// TIA Portal V17 export
// export: Created 2025-03-05T08:02:54.8462086Z, ExportSetting WithDefaults, DisplayName Totally Integrated Automation Portal, DisplayVersion V17 Update 8, DisplayName TIA Portal Openness, DisplayVersion V17 Update 8, DisplayName TIA Portal Version Control Interface, DisplayVersion V17, DisplayName SINAMICS Startdrive Advanced, DisplayVersion V17 SP2, DisplayName SINAMICS Startdrive G110M, G120, G120C, G120D, G120P, G115D, DisplayVersion V17 SP2, DisplayName SINAMICS Startdrive G130, G150, S120, S150, SINAMICS MV, S210, DisplayVersion V17 SP2, DisplayName STEP 7 Professional, DisplayVersion V17 Update 8, DisplayName SINUMERIK ONE STEP 7 Toolbox, DisplayVersion V17 Update 12, DisplayName SINUMERIK 840D sl STEP 7 Toolbox, DisplayVersion V17 Update 12, DisplayName STEP 7 Safety, DisplayVersion V17 Update 6, DisplayName WinCC Advanced, DisplayVersion V17 Update 8
DATA_BLOCK "DB7238_VARIABLES_PLC_CONNECTION"   // DB7238
{ S7_Optimized_Access := 'TRUE'; DB_Accessible_From_OPC_UA := 'FALSE' }
VERSION : 0.1
// stored: AutoNumber false, DBAccessibleFromOPCUA false, DBAccessibleFromWebserver true, IsOnlyStoredInLoadMemory false, IsRetainMemResEnabled false, IsWriteProtectedInAS false, MemoryReserve 100
   VAR RETAIN
      FEEDER_1_U_01_LINE_1 { S7_SetPoint := 'True'} : "UDT_Feeder Line";
      FEEDER_1_U_01_LINE_2 { S7_SetPoint := 'True'} : "UDT_Feeder Line";
      FEEDER_1_U_02_LINE_1 { S7_SetPoint := 'True'} : "UDT_Feeder Line";
      FEEDER_1_U_02_LINE_2 { S7_SetPoint := 'True'} : "UDT_Feeder Line";
      FEEDER_2_U_02_LINE_1 { S7_SetPoint := 'True'} : "UDT_Feeder Line";
      FEEDER_2_U_02_LINE_2 { S7_SetPoint := 'True'} : "UDT_Feeder Line";
      HOPPER_U_01_LINE_1 { S7_SetPoint := 'True'} : "UDT_Hopper Line";
      HOPPER_U_01_LINE_2 { S7_SetPoint := 'True'} : "UDT_Hopper Line";
      HOPPER_U_02_LINE_1 { S7_SetPoint := 'True'} : "UDT_Hopper Line";
      HOPPER_U_02_LINE_2 { S7_SetPoint := 'True'} : "UDT_Hopper Line";
   END_VAR
   VAR
      HOPPER_U_02_LINE_3 { S7_SetPoint := 'True'} : "UDT_Hopper Line";
      GENERAL : Struct
         PLC_TO_HMI : Struct
            FEEDERS_MODE_STATE : Int := 1;   // FEEDERS MODE STATE (1= AUTO. 3= MANUAL)
            HOPPERS_MODE_STATE : Int := 1;   // HOPPERS MODE STATE (1= AUTO. 3= MANUAL)
         END_STRUCT;
         HMI_TO_PLC : Struct
            FEEDERS_AUTO_MODE : Bool := FALSE;   // FEEDERS AUTO MODE HMI BUTTON
            FEEDERS_MANUAL_MODE : Bool := FALSE;   // FEEDERS MANUAL MODE HMI BUTTON
            HOPPERS_AUTO_MODE : Bool := FALSE;   // HOPPERS AUTO MODE HMI BUTTON
            HOPPERS_MANUAL_MODE : Bool := FALSE;   // HOPPERS MANUAL MODE HMI BUTTON
         END_STRUCT;
      END_STRUCT;
   END_VAR
   VAR RETAIN
      SELECTED_UNIT { S7_SetPoint := 'True'} : Int := 0;
      FEEDER_1_U01_SELECTED_GAS : Int := 1;   // SELECTED GAS. 1 = ARGON. 2 = NITROGEN. 3 = HELIUM. 4 = ARGON30
   END_VAR
   VAR
      FEEDER_1_U01_CHANGE_GAS_COND : Bool;   // CHANGE GAS CONDITIONS
   END_VAR
   VAR RETAIN
      FEEDER_1_U02_SELECTED_GAS : Int := 1;   // SELECTED GAS. 1 = ARGON. 2 = NITROGEN. 3 = HELIUM. 4 = ARGON30
   END_VAR
   VAR
      FEEDER_1_U02_CHANGE_GAS_COND : Bool;   // CHANGE GAS CONDITIONS
   END_VAR
   VAR RETAIN
      FEEDER_2_U02_SELECTED_GAS : Int := 1;   // SELECTED GAS. 1 = ARGON. 2 = NITROGEN. 3 = HELIUM. 4 = ARGON30
   END_VAR
   VAR
      FEEDER_2_U02_CHANGE_GAS_COND : Bool;   // CHANGE GAS CONDITIONS
      CURRENT_PROTECTION_LEVEL : Byte := 16#01;   // CURRENT ACCESS LEVEL
      EKS_USER : String := 'ETX4   $07';   // EKS OPERATOR ID
      HMI_USER : String := 'Engineering';
      HMI_PASSWORD : WString := WSTRING#'Engineering';
      EKS_OPERATOR_IDENTIFICATION : Byte := 16#01;   // EKS OPERATOR IDENTIFICATION
   END_VAR
BEGIN
   FEEDER_1_U_01_LINE_1.GAS_FLOW_RATE_ACTUAL := 0.0;
   FEEDER_1_U_01_LINE_1.GAS_FLOW_RATE_AUTO := 11.0;
   FEEDER_1_U_01_LINE_1.GAS_FLOW_RATE_MANUAL := 10.0;
   FEEDER_1_U_01_LINE_1.DISC_SPEED_ACTUAL := 0.0;
   FEEDER_1_U_01_LINE_1.DISC_SPEED_AUTO := 44.0;
   FEEDER_1_U_01_LINE_1.DISC_SPEED_MANUAL := 44.0;
   FEEDER_1_U_01_LINE_1.STIRRER_SPEED_ACTUAL := 0.0;
   FEEDER_1_U_01_LINE_1.STIRRER_SPEED_AUTO := 30.0;
   FEEDER_1_U_01_LINE_1.STIRRER_SPEED_MANUAL := 30.0;
   FEEDER_1_U_01_LINE_1.HOPPER_TEMP_ACTUAL := -1.0;
   FEEDER_1_U_01_LINE_1.HOPPER_TEMP_AUTO := 0.0;
   FEEDER_1_U_01_LINE_1.HOPPER_TEMP_MANUAL := 0.0;
   FEEDER_1_U_01_LINE_1.HEATER_ON_MANUAL_REQUEST := FALSE;
   FEEDER_1_U_01_LINE_1.HEATER_OFF_MANUAL_REQUEST := FALSE;
   FEEDER_1_U_01_LINE_1.HOPPER_ON_MANUAL_REQUEST := FALSE;
   FEEDER_1_U_01_LINE_1.HOPPER_OFF_MANUAL_REQUEST := FALSE;
   FEEDER_1_U_01_LINE_1.HOPPER_STATUS := 16#00;
   FEEDER_1_U_01_LINE_1.START_SEQUENCE_GAS_STEPS := 5;
   FEEDER_1_U_01_LINE_1.START_SEQUENCE_DISK_STEPS := 5;
   FEEDER_1_U_01_LINE_1.STOP_SEQUENCE_GAS_STEPS := 10;
   FEEDER_1_U_01_LINE_1.STOP_SEQUENCE_DISK_STEPS := 10;
   FEEDER_1_U_01_LINE_1.STOP_SEQUENCE_PAUSE_STEP := 5;
   FEEDER_1_U_01_LINE_1.DISC_SPEED_WARNING_UPPER_LIMIT := 1.0;
   FEEDER_1_U_01_LINE_1.DISC_SPEED_ALARM_UPPER_LIMIT := 2.0;
   FEEDER_1_U_01_LINE_1.DISC_SPEED_WARNING_LOWER_LIMIT := 1.0;
   FEEDER_1_U_01_LINE_1.DISC_SPEED_ALARM_LOWER_LIMIT := 2.0;
   FEEDER_1_U_01_LINE_1.GAS_FLOW_RATE_WARNING_UPPER_LIMIT := 1.0;
   FEEDER_1_U_01_LINE_1.GAS_FLOW_RATE_ALARM_UPPER_LIMIT := 4.0;
   FEEDER_1_U_01_LINE_1.GAS_FLOW_RATE_WARNING_LOWER_LIMIT := 1.0;
   FEEDER_1_U_01_LINE_1.GAS_FLOW_RATE_ALARM_LOWER_LIMIT := 4.0;
   FEEDER_1_U_01_LINE_1.STIRRER_SPEED_WARNING_UPPER_LIMIT := 1.0;
   FEEDER_1_U_01_LINE_1.STIRRER_SPEED_ALARM_UPPER_LIMIT := 5.0;
   FEEDER_1_U_01_LINE_1.STIRRER_SPEED_WARNING_LOWER_LIMIT := 1.0;
   FEEDER_1_U_01_LINE_1.STIRRER_SPEED_ALARM_LOWER_LIMIT := 10.0;
   FEEDER_1_U_01_LINE_1.HOPPER_TEMP_ALARM_UPPER_LIMIT := 3.0;
   FEEDER_1_U_01_LINE_1.PRESSURE_VALUE_CURRENT_SENSOR := 0.0;
   FEEDER_1_U_01_LINE_2.GAS_FLOW_RATE_ACTUAL := 0.0;
   FEEDER_1_U_01_LINE_2.GAS_FLOW_RATE_AUTO := 11.0;
   FEEDER_1_U_01_LINE_2.GAS_FLOW_RATE_MANUAL := 10.0;
   FEEDER_1_U_01_LINE_2.DISC_SPEED_ACTUAL := 0.0;
   FEEDER_1_U_01_LINE_2.DISC_SPEED_AUTO := 44.0;
   FEEDER_1_U_01_LINE_2.DISC_SPEED_MANUAL := 44.0;
   FEEDER_1_U_01_LINE_2.STIRRER_SPEED_ACTUAL := 0.0;
   FEEDER_1_U_01_LINE_2.STIRRER_SPEED_AUTO := 30.0;
   FEEDER_1_U_01_LINE_2.STIRRER_SPEED_MANUAL := 30.0;
   FEEDER_1_U_01_LINE_2.HOPPER_TEMP_ACTUAL := -1.0;
   FEEDER_1_U_01_LINE_2.HOPPER_TEMP_AUTO := 0.0;
   FEEDER_1_U_01_LINE_2.HOPPER_TEMP_MANUAL := 0.0;
   FEEDER_1_U_01_LINE_2.HEATER_ON_MANUAL_REQUEST := FALSE;
   FEEDER_1_U_01_LINE_2.HEATER_OFF_MANUAL_REQUEST := FALSE;
   FEEDER_1_U_01_LINE_2.HOPPER_ON_MANUAL_REQUEST := FALSE;
   FEEDER_1_U_01_LINE_2.HOPPER_OFF_MANUAL_REQUEST := FALSE;
   FEEDER_1_U_01_LINE_2.HOPPER_STATUS := 16#00;
   FEEDER_1_U_01_LINE_2.START_SEQUENCE_GAS_STEPS := 5;
   FEEDER_1_U_01_LINE_2.START_SEQUENCE_DISK_STEPS := 5;
   FEEDER_1_U_01_LINE_2.STOP_SEQUENCE_GAS_STEPS := 10;
   FEEDER_1_U_01_LINE_2.STOP_SEQUENCE_DISK_STEPS := 10;
   FEEDER_1_U_01_LINE_2.STOP_SEQUENCE_PAUSE_STEP := 5;
   FEEDER_1_U_01_LINE_2.DISC_SPEED_WARNING_UPPER_LIMIT := 1.0;
   FEEDER_1_U_01_LINE_2.DISC_SPEED_ALARM_UPPER_LIMIT := 2.0;
   FEEDER_1_U_01_LINE_2.DISC_SPEED_WARNING_LOWER_LIMIT := 1.0;
   FEEDER_1_U_01_LINE_2.DISC_SPEED_ALARM_LOWER_LIMIT := 2.0;
   FEEDER_1_U_01_LINE_2.GAS_FLOW_RATE_WARNING_UPPER_LIMIT := 1.0;
   FEEDER_1_U_01_LINE_2.GAS_FLOW_RATE_ALARM_UPPER_LIMIT := 4.0;
   FEEDER_1_U_01_LINE_2.GAS_FLOW_RATE_WARNING_LOWER_LIMIT := 1.0;
   FEEDER_1_U_01_LINE_2.GAS_FLOW_RATE_ALARM_LOWER_LIMIT := 4.0;
   FEEDER_1_U_01_LINE_2.STIRRER_SPEED_WARNING_UPPER_LIMIT := 1.0;
   FEEDER_1_U_01_LINE_2.STIRRER_SPEED_ALARM_UPPER_LIMIT := 5.0;
   FEEDER_1_U_01_LINE_2.STIRRER_SPEED_WARNING_LOWER_LIMIT := 1.0;
   FEEDER_1_U_01_LINE_2.STIRRER_SPEED_ALARM_LOWER_LIMIT := 10.0;
   FEEDER_1_U_01_LINE_2.HOPPER_TEMP_ALARM_UPPER_LIMIT := 3.0;
   FEEDER_1_U_01_LINE_2.PRESSURE_VALUE_CURRENT_SENSOR := 0.0;
   FEEDER_1_U_02_LINE_1.GAS_FLOW_RATE_ACTUAL := 13.99967;
   FEEDER_1_U_02_LINE_1.GAS_FLOW_RATE_AUTO := 14.0;
   FEEDER_1_U_02_LINE_1.GAS_FLOW_RATE_MANUAL := 14.0;
   FEEDER_1_U_02_LINE_1.DISC_SPEED_ACTUAL := 78.12334;
   FEEDER_1_U_02_LINE_1.DISC_SPEED_AUTO := 78.0;
   FEEDER_1_U_02_LINE_1.DISC_SPEED_MANUAL := 77.0;
   FEEDER_1_U_02_LINE_1.STIRRER_SPEED_ACTUAL := 30.15667;
   FEEDER_1_U_02_LINE_1.STIRRER_SPEED_AUTO := 30.0;
   FEEDER_1_U_02_LINE_1.STIRRER_SPEED_MANUAL := 30.0;
   FEEDER_1_U_02_LINE_1.HOPPER_TEMP_ACTUAL := 17.4;
   FEEDER_1_U_02_LINE_1.HOPPER_TEMP_AUTO := 0.0;
   FEEDER_1_U_02_LINE_1.HOPPER_TEMP_MANUAL := 0.0;
   FEEDER_1_U_02_LINE_1.HEATER_ON_MANUAL_REQUEST := FALSE;
   FEEDER_1_U_02_LINE_1.HEATER_OFF_MANUAL_REQUEST := FALSE;
   FEEDER_1_U_02_LINE_1.HOPPER_ON_MANUAL_REQUEST := FALSE;
   FEEDER_1_U_02_LINE_1.HOPPER_OFF_MANUAL_REQUEST := FALSE;
   FEEDER_1_U_02_LINE_1.HOPPER_STATUS := 16#01;
   FEEDER_1_U_02_LINE_1.START_SEQUENCE_GAS_STEPS := 5;
   FEEDER_1_U_02_LINE_1.START_SEQUENCE_DISK_STEPS := 5;
   FEEDER_1_U_02_LINE_1.STOP_SEQUENCE_GAS_STEPS := 10;
   FEEDER_1_U_02_LINE_1.STOP_SEQUENCE_DISK_STEPS := 10;
   FEEDER_1_U_02_LINE_1.STOP_SEQUENCE_PAUSE_STEP := 5;
   FEEDER_1_U_02_LINE_1.DISC_SPEED_WARNING_UPPER_LIMIT := 10.0;
   FEEDER_1_U_02_LINE_1.DISC_SPEED_ALARM_UPPER_LIMIT := 2.0;
   FEEDER_1_U_02_LINE_1.DISC_SPEED_WARNING_LOWER_LIMIT := 15.0;
   FEEDER_1_U_02_LINE_1.DISC_SPEED_ALARM_LOWER_LIMIT := 2.0;
   FEEDER_1_U_02_LINE_1.GAS_FLOW_RATE_WARNING_UPPER_LIMIT := 3.0;
   FEEDER_1_U_02_LINE_1.GAS_FLOW_RATE_ALARM_UPPER_LIMIT := 4.0;
   FEEDER_1_U_02_LINE_1.GAS_FLOW_RATE_WARNING_LOWER_LIMIT := 15.0;
   FEEDER_1_U_02_LINE_1.GAS_FLOW_RATE_ALARM_LOWER_LIMIT := 4.0;
   FEEDER_1_U_02_LINE_1.STIRRER_SPEED_WARNING_UPPER_LIMIT := 10.0;
   FEEDER_1_U_02_LINE_1.STIRRER_SPEED_ALARM_UPPER_LIMIT := 5.0;
   FEEDER_1_U_02_LINE_1.STIRRER_SPEED_WARNING_LOWER_LIMIT := 99.0;
   FEEDER_1_U_02_LINE_1.STIRRER_SPEED_ALARM_LOWER_LIMIT := 10.0;
   FEEDER_1_U_02_LINE_1.HOPPER_TEMP_ALARM_UPPER_LIMIT := 0.0;
   FEEDER_1_U_02_LINE_1.PRESSURE_VALUE_CURRENT_SENSOR := 0.0;
   FEEDER_1_U_02_LINE_2.GAS_FLOW_RATE_ACTUAL := 13.99837;
   FEEDER_1_U_02_LINE_2.GAS_FLOW_RATE_AUTO := 14.0;
   FEEDER_1_U_02_LINE_2.GAS_FLOW_RATE_MANUAL := 14.0;
   FEEDER_1_U_02_LINE_2.DISC_SPEED_ACTUAL := 77.98333;
   FEEDER_1_U_02_LINE_2.DISC_SPEED_AUTO := 78.0;
   FEEDER_1_U_02_LINE_2.DISC_SPEED_MANUAL := 77.0;
   FEEDER_1_U_02_LINE_2.STIRRER_SPEED_ACTUAL := 29.89333;
   FEEDER_1_U_02_LINE_2.STIRRER_SPEED_AUTO := 30.0;
   FEEDER_1_U_02_LINE_2.STIRRER_SPEED_MANUAL := 30.0;
   FEEDER_1_U_02_LINE_2.HOPPER_TEMP_ACTUAL := 17.6;
   FEEDER_1_U_02_LINE_2.HOPPER_TEMP_AUTO := 0.0;
   FEEDER_1_U_02_LINE_2.HOPPER_TEMP_MANUAL := 0.0;
   FEEDER_1_U_02_LINE_2.HEATER_ON_MANUAL_REQUEST := FALSE;
   FEEDER_1_U_02_LINE_2.HEATER_OFF_MANUAL_REQUEST := FALSE;
   FEEDER_1_U_02_LINE_2.HOPPER_ON_MANUAL_REQUEST := FALSE;
   FEEDER_1_U_02_LINE_2.HOPPER_OFF_MANUAL_REQUEST := FALSE;
   FEEDER_1_U_02_LINE_2.HOPPER_STATUS := 16#01;
   FEEDER_1_U_02_LINE_2.START_SEQUENCE_GAS_STEPS := 5;
   FEEDER_1_U_02_LINE_2.START_SEQUENCE_DISK_STEPS := 5;
   FEEDER_1_U_02_LINE_2.STOP_SEQUENCE_GAS_STEPS := 10;
   FEEDER_1_U_02_LINE_2.STOP_SEQUENCE_DISK_STEPS := 10;
   FEEDER_1_U_02_LINE_2.STOP_SEQUENCE_PAUSE_STEP := 5;
   FEEDER_1_U_02_LINE_2.DISC_SPEED_WARNING_UPPER_LIMIT := 10.0;
   FEEDER_1_U_02_LINE_2.DISC_SPEED_ALARM_UPPER_LIMIT := 2.0;
   FEEDER_1_U_02_LINE_2.DISC_SPEED_WARNING_LOWER_LIMIT := 15.0;
   FEEDER_1_U_02_LINE_2.DISC_SPEED_ALARM_LOWER_LIMIT := 2.0;
   FEEDER_1_U_02_LINE_2.GAS_FLOW_RATE_WARNING_UPPER_LIMIT := 3.0;
   FEEDER_1_U_02_LINE_2.GAS_FLOW_RATE_ALARM_UPPER_LIMIT := 4.0;
   FEEDER_1_U_02_LINE_2.GAS_FLOW_RATE_WARNING_LOWER_LIMIT := 15.0;
   FEEDER_1_U_02_LINE_2.GAS_FLOW_RATE_ALARM_LOWER_LIMIT := 4.0;
   FEEDER_1_U_02_LINE_2.STIRRER_SPEED_WARNING_UPPER_LIMIT := 10.0;
   FEEDER_1_U_02_LINE_2.STIRRER_SPEED_ALARM_UPPER_LIMIT := 5.0;
   FEEDER_1_U_02_LINE_2.STIRRER_SPEED_WARNING_LOWER_LIMIT := 99.0;
   FEEDER_1_U_02_LINE_2.STIRRER_SPEED_ALARM_LOWER_LIMIT := 10.0;
   FEEDER_1_U_02_LINE_2.HOPPER_TEMP_ALARM_UPPER_LIMIT := 3.0;
   FEEDER_1_U_02_LINE_2.PRESSURE_VALUE_CURRENT_SENSOR := 0.0;
   FEEDER_2_U_02_LINE_1.GAS_FLOW_RATE_ACTUAL := 0.0;
   FEEDER_2_U_02_LINE_1.GAS_FLOW_RATE_AUTO := 0.0;
   FEEDER_2_U_02_LINE_1.GAS_FLOW_RATE_MANUAL := 0.0;
   FEEDER_2_U_02_LINE_1.DISC_SPEED_ACTUAL := 0.0;
   FEEDER_2_U_02_LINE_1.DISC_SPEED_AUTO := 0.0;
   FEEDER_2_U_02_LINE_1.DISC_SPEED_MANUAL := 0.0;
   FEEDER_2_U_02_LINE_1.STIRRER_SPEED_ACTUAL := 0.0;
   FEEDER_2_U_02_LINE_1.STIRRER_SPEED_AUTO := 0.0;
   FEEDER_2_U_02_LINE_1.STIRRER_SPEED_MANUAL := 0.0;
   FEEDER_2_U_02_LINE_1.HOPPER_TEMP_ACTUAL := 0.0;
   FEEDER_2_U_02_LINE_1.HOPPER_TEMP_AUTO := 0.0;
   FEEDER_2_U_02_LINE_1.HOPPER_TEMP_MANUAL := 0.0;
   FEEDER_2_U_02_LINE_1.HEATER_ON_MANUAL_REQUEST := FALSE;
   FEEDER_2_U_02_LINE_1.HEATER_OFF_MANUAL_REQUEST := FALSE;
   FEEDER_2_U_02_LINE_1.HOPPER_ON_MANUAL_REQUEST := FALSE;
   FEEDER_2_U_02_LINE_1.HOPPER_OFF_MANUAL_REQUEST := FALSE;
   FEEDER_2_U_02_LINE_1.HOPPER_STATUS := 16#00;
   FEEDER_2_U_02_LINE_1.START_SEQUENCE_GAS_STEPS := 0;
   FEEDER_2_U_02_LINE_1.START_SEQUENCE_DISK_STEPS := 0;
   FEEDER_2_U_02_LINE_1.STOP_SEQUENCE_GAS_STEPS := 0;
   FEEDER_2_U_02_LINE_1.STOP_SEQUENCE_DISK_STEPS := 0;
   FEEDER_2_U_02_LINE_1.STOP_SEQUENCE_PAUSE_STEP := 0;
   FEEDER_2_U_02_LINE_1.DISC_SPEED_WARNING_UPPER_LIMIT := 0.0;
   FEEDER_2_U_02_LINE_1.DISC_SPEED_ALARM_UPPER_LIMIT := 0.0;
   FEEDER_2_U_02_LINE_1.DISC_SPEED_WARNING_LOWER_LIMIT := 0.0;
   FEEDER_2_U_02_LINE_1.DISC_SPEED_ALARM_LOWER_LIMIT := 0.0;
   FEEDER_2_U_02_LINE_1.GAS_FLOW_RATE_WARNING_UPPER_LIMIT := 0.0;
   FEEDER_2_U_02_LINE_1.GAS_FLOW_RATE_ALARM_UPPER_LIMIT := 0.0;
   FEEDER_2_U_02_LINE_1.GAS_FLOW_RATE_WARNING_LOWER_LIMIT := 0.0;
   FEEDER_2_U_02_LINE_1.GAS_FLOW_RATE_ALARM_LOWER_LIMIT := 0.0;
   FEEDER_2_U_02_LINE_1.STIRRER_SPEED_WARNING_UPPER_LIMIT := 0.0;
   FEEDER_2_U_02_LINE_1.STIRRER_SPEED_ALARM_UPPER_LIMIT := 0.0;
   FEEDER_2_U_02_LINE_1.STIRRER_SPEED_WARNING_LOWER_LIMIT := 0.0;
   FEEDER_2_U_02_LINE_1.STIRRER_SPEED_ALARM_LOWER_LIMIT := 0.0;
   FEEDER_2_U_02_LINE_1.HOPPER_TEMP_ALARM_UPPER_LIMIT := 0.0;
   FEEDER_2_U_02_LINE_1.PRESSURE_VALUE_CURRENT_SENSOR := 0.0;
   FEEDER_2_U_02_LINE_2.GAS_FLOW_RATE_ACTUAL := 14.00755;
   FEEDER_2_U_02_LINE_2.GAS_FLOW_RATE_AUTO := 14.0;
   FEEDER_2_U_02_LINE_2.GAS_FLOW_RATE_MANUAL := 14.0;
   FEEDER_2_U_02_LINE_2.DISC_SPEED_ACTUAL := 44.02667;
   FEEDER_2_U_02_LINE_2.DISC_SPEED_AUTO := 44.0;
   FEEDER_2_U_02_LINE_2.DISC_SPEED_MANUAL := 77.0;
   FEEDER_2_U_02_LINE_2.STIRRER_SPEED_ACTUAL := 29.94667;
   FEEDER_2_U_02_LINE_2.STIRRER_SPEED_AUTO := 30.0;
   FEEDER_2_U_02_LINE_2.STIRRER_SPEED_MANUAL := 30.0;
   FEEDER_2_U_02_LINE_2.HOPPER_TEMP_ACTUAL := 17.4;
   FEEDER_2_U_02_LINE_2.HOPPER_TEMP_AUTO := 0.0;
   FEEDER_2_U_02_LINE_2.HOPPER_TEMP_MANUAL := 0.0;
   FEEDER_2_U_02_LINE_2.HEATER_ON_MANUAL_REQUEST := FALSE;
   FEEDER_2_U_02_LINE_2.HEATER_OFF_MANUAL_REQUEST := FALSE;
   FEEDER_2_U_02_LINE_2.HOPPER_ON_MANUAL_REQUEST := FALSE;
   FEEDER_2_U_02_LINE_2.HOPPER_OFF_MANUAL_REQUEST := FALSE;
   FEEDER_2_U_02_LINE_2.HOPPER_STATUS := 16#01;
   FEEDER_2_U_02_LINE_2.START_SEQUENCE_GAS_STEPS := 5;
   FEEDER_2_U_02_LINE_2.START_SEQUENCE_DISK_STEPS := 5;
   FEEDER_2_U_02_LINE_2.STOP_SEQUENCE_GAS_STEPS := 10;
   FEEDER_2_U_02_LINE_2.STOP_SEQUENCE_DISK_STEPS := 10;
   FEEDER_2_U_02_LINE_2.STOP_SEQUENCE_PAUSE_STEP := 5;
   FEEDER_2_U_02_LINE_2.DISC_SPEED_WARNING_UPPER_LIMIT := 10.0;
   FEEDER_2_U_02_LINE_2.DISC_SPEED_ALARM_UPPER_LIMIT := 2.0;
   FEEDER_2_U_02_LINE_2.DISC_SPEED_WARNING_LOWER_LIMIT := 15.0;
   FEEDER_2_U_02_LINE_2.DISC_SPEED_ALARM_LOWER_LIMIT := 2.0;
   FEEDER_2_U_02_LINE_2.GAS_FLOW_RATE_WARNING_UPPER_LIMIT := 3.0;
   FEEDER_2_U_02_LINE_2.GAS_FLOW_RATE_ALARM_UPPER_LIMIT := 4.0;
   FEEDER_2_U_02_LINE_2.GAS_FLOW_RATE_WARNING_LOWER_LIMIT := 15.0;
   FEEDER_2_U_02_LINE_2.GAS_FLOW_RATE_ALARM_LOWER_LIMIT := 4.0;
   FEEDER_2_U_02_LINE_2.STIRRER_SPEED_WARNING_UPPER_LIMIT := 10.0;
   FEEDER_2_U_02_LINE_2.STIRRER_SPEED_ALARM_UPPER_LIMIT := 5.0;
   FEEDER_2_U_02_LINE_2.STIRRER_SPEED_WARNING_LOWER_LIMIT := 99.0;
   FEEDER_2_U_02_LINE_2.STIRRER_SPEED_ALARM_LOWER_LIMIT := 10.0;
   FEEDER_2_U_02_LINE_2.HOPPER_TEMP_ALARM_UPPER_LIMIT := 3.0;
   FEEDER_2_U_02_LINE_2.PRESSURE_VALUE_CURRENT_SENSOR := 0.0;
   HOPPER_U_01_LINE_1.STIRRER_SPEED_ACTUAL := 0;
   HOPPER_U_01_LINE_1.STIRRER_SPEED_MANUAL := 0;
   HOPPER_U_01_LINE_1.STIRRER_SPEED_AUTO := 0;
   HOPPER_U_01_LINE_1.TEMP_UPPER_JACKET_ACTUAL := 0.0;
   HOPPER_U_01_LINE_1.TEMP_UPPER_JACKET_MANUAL := 0.0;
   HOPPER_U_01_LINE_1.TEMP_UPPER_JACKET_AUTO := 0.0;
   HOPPER_U_01_LINE_1.TEMP_LOWER_JACKET_ACTUAL := 0.0;
   HOPPER_U_01_LINE_1.TEMP_LOWER_JACKET_MANUAL := 0.0;
   HOPPER_U_01_LINE_1.TEMP_LOWER_JACKET_AUTO := 0.0;
   HOPPER_U_01_LINE_1.MAX_WEIGHT_ACTUAL := 0.0;
   HOPPER_U_01_LINE_1.MAX_WEIGHT_MANUAL := 0.0;
   HOPPER_U_01_LINE_1.TOTAL_WEIGHT_ACTUAL := 0.0;
   HOPPER_U_01_LINE_1.HOPPER_WEIGHT_ACTUAL := 0.0;
   HOPPER_U_01_LINE_1.HOPPER_WEIGHT_MANUAL := 0.0;
   HOPPER_U_01_LINE_1.POWDER_WEIGHT_ACTUAL := 0.0;
   HOPPER_U_01_LINE_1.HOPPER_COVER_ACTUAL := 0.0;
   HOPPER_U_01_LINE_1.HOPPER_COVER_MANUAL := 0.0;
   HOPPER_U_01_LINE_1.HOPPER_COVER_AUTO := 0.0;
   HOPPER_U_01_LINE_1.FEEDING_COVER_ACTUAL := 0.0;
   HOPPER_U_01_LINE_1.FEEDER_DISK_PRESSURE_ACTUAL := 0.0;
   HOPPER_U_01_LINE_1.TRANSFER_POWDER_SEQ_START := FALSE;
   HOPPER_U_01_LINE_1.TRANSFER_POWDER_SEQ_STOP := FALSE;
   HOPPER_U_01_LINE_1.PRESSURIZE_GAS_VALVE_START := FALSE;
   HOPPER_U_01_LINE_1.PRESSURIZE_GAS_VALVE_STOP := FALSE;
   HOPPER_U_01_LINE_1.RELIEVE_GAS_VALVE_START := FALSE;
   HOPPER_U_01_LINE_1.RELIEVE_GAS_VALVE_STOP := FALSE;
   HOPPER_U_01_LINE_1.CLEANING_AIR_VALVE_START := FALSE;
   HOPPER_U_01_LINE_1.CLEANING_AIR_VALVE_STOP := FALSE;
   HOPPER_U_01_LINE_1.LOAD_FEEDER_SEQUENCE_START := FALSE;
   HOPPER_U_01_LINE_1.LOAD_FEEDER_SEQUENCE_STOP := FALSE;
   HOPPER_U_01_LINE_2.STIRRER_SPEED_ACTUAL := 0;
   HOPPER_U_01_LINE_2.STIRRER_SPEED_MANUAL := 25;
   HOPPER_U_01_LINE_2.STIRRER_SPEED_AUTO := 0;
   HOPPER_U_01_LINE_2.TEMP_UPPER_JACKET_ACTUAL := 0.0;
   HOPPER_U_01_LINE_2.TEMP_UPPER_JACKET_MANUAL := 0.0;
   HOPPER_U_01_LINE_2.TEMP_UPPER_JACKET_AUTO := 0.0;
   HOPPER_U_01_LINE_2.TEMP_LOWER_JACKET_ACTUAL := 0.0;
   HOPPER_U_01_LINE_2.TEMP_LOWER_JACKET_MANUAL := 0.0;
   HOPPER_U_01_LINE_2.TEMP_LOWER_JACKET_AUTO := 0.0;
   HOPPER_U_01_LINE_2.MAX_WEIGHT_ACTUAL := 0.0;
   HOPPER_U_01_LINE_2.MAX_WEIGHT_MANUAL := 0.0;
   HOPPER_U_01_LINE_2.TOTAL_WEIGHT_ACTUAL := 0.0;
   HOPPER_U_01_LINE_2.HOPPER_WEIGHT_ACTUAL := 0.0;
   HOPPER_U_01_LINE_2.HOPPER_WEIGHT_MANUAL := 0.0;
   HOPPER_U_01_LINE_2.POWDER_WEIGHT_ACTUAL := 0.0;
   HOPPER_U_01_LINE_2.HOPPER_COVER_ACTUAL := 0.0;
   HOPPER_U_01_LINE_2.HOPPER_COVER_MANUAL := 0.0;
   HOPPER_U_01_LINE_2.HOPPER_COVER_AUTO := 0.0;
   HOPPER_U_01_LINE_2.FEEDING_COVER_ACTUAL := 0.0;
   HOPPER_U_01_LINE_2.FEEDER_DISK_PRESSURE_ACTUAL := 0.0;
   HOPPER_U_01_LINE_2.TRANSFER_POWDER_SEQ_START := FALSE;
   HOPPER_U_01_LINE_2.TRANSFER_POWDER_SEQ_STOP := FALSE;
   HOPPER_U_01_LINE_2.PRESSURIZE_GAS_VALVE_START := FALSE;
   HOPPER_U_01_LINE_2.PRESSURIZE_GAS_VALVE_STOP := FALSE;
   HOPPER_U_01_LINE_2.RELIEVE_GAS_VALVE_START := FALSE;
   HOPPER_U_01_LINE_2.RELIEVE_GAS_VALVE_STOP := FALSE;
   HOPPER_U_01_LINE_2.CLEANING_AIR_VALVE_START := FALSE;
   HOPPER_U_01_LINE_2.CLEANING_AIR_VALVE_STOP := FALSE;
   HOPPER_U_01_LINE_2.LOAD_FEEDER_SEQUENCE_START := FALSE;
   HOPPER_U_01_LINE_2.LOAD_FEEDER_SEQUENCE_STOP := FALSE;
   HOPPER_U_02_LINE_1.STIRRER_SPEED_ACTUAL := 0;
   HOPPER_U_02_LINE_1.STIRRER_SPEED_MANUAL := 0;
   HOPPER_U_02_LINE_1.STIRRER_SPEED_AUTO := 0;
   HOPPER_U_02_LINE_1.TEMP_UPPER_JACKET_ACTUAL := 0.0;
   HOPPER_U_02_LINE_1.TEMP_UPPER_JACKET_MANUAL := 0.0;
   HOPPER_U_02_LINE_1.TEMP_UPPER_JACKET_AUTO := 0.0;
   HOPPER_U_02_LINE_1.TEMP_LOWER_JACKET_ACTUAL := 0.0;
   HOPPER_U_02_LINE_1.TEMP_LOWER_JACKET_MANUAL := 0.0;
   HOPPER_U_02_LINE_1.TEMP_LOWER_JACKET_AUTO := 0.0;
   HOPPER_U_02_LINE_1.MAX_WEIGHT_ACTUAL := 0.0;
   HOPPER_U_02_LINE_1.MAX_WEIGHT_MANUAL := 0.0;
   HOPPER_U_02_LINE_1.TOTAL_WEIGHT_ACTUAL := 0.0;
   HOPPER_U_02_LINE_1.HOPPER_WEIGHT_ACTUAL := 0.0;
   HOPPER_U_02_LINE_1.HOPPER_WEIGHT_MANUAL := 0.0;
   HOPPER_U_02_LINE_1.POWDER_WEIGHT_ACTUAL := 0.0;
   HOPPER_U_02_LINE_1.HOPPER_COVER_ACTUAL := 0.0;
   HOPPER_U_02_LINE_1.HOPPER_COVER_MANUAL := 0.0;
   HOPPER_U_02_LINE_1.HOPPER_COVER_AUTO := 0.0;
   HOPPER_U_02_LINE_1.FEEDING_COVER_ACTUAL := 0.0;
   HOPPER_U_02_LINE_1.FEEDER_DISK_PRESSURE_ACTUAL := 0.0;
   HOPPER_U_02_LINE_1.TRANSFER_POWDER_SEQ_START := FALSE;
   HOPPER_U_02_LINE_1.TRANSFER_POWDER_SEQ_STOP := FALSE;
   HOPPER_U_02_LINE_1.PRESSURIZE_GAS_VALVE_START := FALSE;
   HOPPER_U_02_LINE_1.PRESSURIZE_GAS_VALVE_STOP := FALSE;
   HOPPER_U_02_LINE_1.RELIEVE_GAS_VALVE_START := FALSE;
   HOPPER_U_02_LINE_1.RELIEVE_GAS_VALVE_STOP := FALSE;
   HOPPER_U_02_LINE_1.CLEANING_AIR_VALVE_START := FALSE;
   HOPPER_U_02_LINE_1.CLEANING_AIR_VALVE_STOP := FALSE;
   HOPPER_U_02_LINE_1.LOAD_FEEDER_SEQUENCE_START := FALSE;
   HOPPER_U_02_LINE_1.LOAD_FEEDER_SEQUENCE_STOP := FALSE;
   HOPPER_U_02_LINE_2.STIRRER_SPEED_ACTUAL := 0;
   HOPPER_U_02_LINE_2.STIRRER_SPEED_MANUAL := 0;
   HOPPER_U_02_LINE_2.STIRRER_SPEED_AUTO := 0;
   HOPPER_U_02_LINE_2.TEMP_UPPER_JACKET_ACTUAL := 0.0;
   HOPPER_U_02_LINE_2.TEMP_UPPER_JACKET_MANUAL := 0.0;
   HOPPER_U_02_LINE_2.TEMP_UPPER_JACKET_AUTO := 0.0;
   HOPPER_U_02_LINE_2.TEMP_LOWER_JACKET_ACTUAL := 0.0;
   HOPPER_U_02_LINE_2.TEMP_LOWER_JACKET_MANUAL := 0.0;
   HOPPER_U_02_LINE_2.TEMP_LOWER_JACKET_AUTO := 0.0;
   HOPPER_U_02_LINE_2.MAX_WEIGHT_ACTUAL := 0.0;
   HOPPER_U_02_LINE_2.MAX_WEIGHT_MANUAL := 0.0;
   HOPPER_U_02_LINE_2.TOTAL_WEIGHT_ACTUAL := 0.0;
   HOPPER_U_02_LINE_2.HOPPER_WEIGHT_ACTUAL := 0.0;
   HOPPER_U_02_LINE_2.HOPPER_WEIGHT_MANUAL := 0.0;
   HOPPER_U_02_LINE_2.POWDER_WEIGHT_ACTUAL := 0.0;
   HOPPER_U_02_LINE_2.HOPPER_COVER_ACTUAL := 0.0;
   HOPPER_U_02_LINE_2.HOPPER_COVER_MANUAL := 0.0;
   HOPPER_U_02_LINE_2.HOPPER_COVER_AUTO := 0.0;
   HOPPER_U_02_LINE_2.FEEDING_COVER_ACTUAL := 0.0;
   HOPPER_U_02_LINE_2.FEEDER_DISK_PRESSURE_ACTUAL := 0.0;
   HOPPER_U_02_LINE_2.TRANSFER_POWDER_SEQ_START := FALSE;
   HOPPER_U_02_LINE_2.TRANSFER_POWDER_SEQ_STOP := FALSE;
   HOPPER_U_02_LINE_2.PRESSURIZE_GAS_VALVE_START := FALSE;
   HOPPER_U_02_LINE_2.PRESSURIZE_GAS_VALVE_STOP := FALSE;
   HOPPER_U_02_LINE_2.RELIEVE_GAS_VALVE_START := FALSE;
   HOPPER_U_02_LINE_2.RELIEVE_GAS_VALVE_STOP := FALSE;
   HOPPER_U_02_LINE_2.CLEANING_AIR_VALVE_START := FALSE;
   HOPPER_U_02_LINE_2.CLEANING_AIR_VALVE_STOP := FALSE;
   HOPPER_U_02_LINE_2.LOAD_FEEDER_SEQUENCE_START := FALSE;
   HOPPER_U_02_LINE_2.LOAD_FEEDER_SEQUENCE_STOP := FALSE;
   HOPPER_U_02_LINE_3.STIRRER_SPEED_ACTUAL := 0;
   HOPPER_U_02_LINE_3.STIRRER_SPEED_MANUAL := 0;
   HOPPER_U_02_LINE_3.STIRRER_SPEED_AUTO := 0;
   HOPPER_U_02_LINE_3.TEMP_UPPER_JACKET_ACTUAL := 0.0;
   HOPPER_U_02_LINE_3.TEMP_UPPER_JACKET_MANUAL := 0.0;
   HOPPER_U_02_LINE_3.TEMP_UPPER_JACKET_AUTO := 0.0;
   HOPPER_U_02_LINE_3.TEMP_LOWER_JACKET_ACTUAL := 0.0;
   HOPPER_U_02_LINE_3.TEMP_LOWER_JACKET_MANUAL := 0.0;
   HOPPER_U_02_LINE_3.TEMP_LOWER_JACKET_AUTO := 0.0;
   HOPPER_U_02_LINE_3.MAX_WEIGHT_ACTUAL := 0.0;
   HOPPER_U_02_LINE_3.MAX_WEIGHT_MANUAL := 0.0;
   HOPPER_U_02_LINE_3.TOTAL_WEIGHT_ACTUAL := 0.0;
   HOPPER_U_02_LINE_3.HOPPER_WEIGHT_ACTUAL := 0.0;
   HOPPER_U_02_LINE_3.HOPPER_WEIGHT_MANUAL := 0.0;
   HOPPER_U_02_LINE_3.POWDER_WEIGHT_ACTUAL := 0.0;
   HOPPER_U_02_LINE_3.HOPPER_COVER_ACTUAL := 0.0;
   HOPPER_U_02_LINE_3.HOPPER_COVER_MANUAL := 0.0;
   HOPPER_U_02_LINE_3.HOPPER_COVER_AUTO := 0.0;
   HOPPER_U_02_LINE_3.FEEDING_COVER_ACTUAL := 0.0;
   HOPPER_U_02_LINE_3.FEEDER_DISK_PRESSURE_ACTUAL := 0.0;
   HOPPER_U_02_LINE_3.TRANSFER_POWDER_SEQ_START := FALSE;
   HOPPER_U_02_LINE_3.TRANSFER_POWDER_SEQ_STOP := FALSE;
   HOPPER_U_02_LINE_3.PRESSURIZE_GAS_VALVE_START := FALSE;
   HOPPER_U_02_LINE_3.PRESSURIZE_GAS_VALVE_STOP := FALSE;
   HOPPER_U_02_LINE_3.RELIEVE_GAS_VALVE_START := FALSE;
   HOPPER_U_02_LINE_3.RELIEVE_GAS_VALVE_STOP := FALSE;
   HOPPER_U_02_LINE_3.CLEANING_AIR_VALVE_START := FALSE;
   HOPPER_U_02_LINE_3.CLEANING_AIR_VALVE_STOP := FALSE;
   HOPPER_U_02_LINE_3.LOAD_FEEDER_SEQUENCE_START := FALSE;
   HOPPER_U_02_LINE_3.LOAD_FEEDER_SEQUENCE_STOP := FALSE;
END_DATA_BLOCK
